FUNCTION_BLOCK StartProgramTask EXTENDS TcoUrRoboticsTask
VAR

	_stopType: TcoAbstractions.eTcoRoboticsStopType;
END_VAR



IF Execute() THEN
	_blink(inOnTime:=T#500MS,inOffTime:=T#500MS);

	IF _progress = 0 THEN
		IF NOT __ISVALIDREF(inoControl) THEN
			_varInfo :=__VARINFO(inoControl);
			Messenger.Programming(_sb.Clear().Append('<#Invalid reference: #>').Append(_varInfo.Symbol).ToString()).Pin();
		ELSIF NOT __ISVALIDREF(inoConfig) THEN                                                  
			_varInfo :=__VARINFO(inoConfig);                                                    
			Messenger.Programming(_sb.Clear().Append('<#Invalid reference: #>').Append(_varInfo.Symbol).ToString()).Pin();
		ELSIF NOT __ISVALIDREF(inoStatus) THEN                                                  
			_varInfo :=__VARINFO(inoStatus);                                                    
			Messenger.Programming(_sb.Clear().Append('<#Invalid reference: #>').Append(_varInfo.Symbol).ToString()).Pin();
			ELSE
			_progress := _progress + 1;
		END_IF

	END_IF
	IF _progress = 1 THEN
		inoControl.StartProgram:=_blink.outQ;
		_varInfo :=__VARINFO( inoStatus.State.CycleOn);                                                
		THIS^.Messenger.OnCondition(_infoTimer.Q AND NOT inoStatus.State.CycleOn).Warning(_sb.Clear().Append('<#Waiting for program running signal! #>').Append(_varInfo.Symbol).ToString());
		
		_varInfo :=__VARINFO( inoStatus.State.SystemInputBusy);                                                
		THIS^.Messenger.OnCondition(_infoTimer.Q AND  inoStatus.State.SystemInputBusy).Warning(_sb.Clear().Append('<#Waiting for system ready signal! #>').Append(_varInfo.Symbol).ToString());
		
		IF  inoStatus.State.CycleOn AND NOT inoStatus.State.SystemInputBusy THEN
				inoControl.StartProgram:=FALSE;
		END_IF
	END_IF;		
	
	

    DoneWhen(inoStatus.State.CycleOn );
    CallTimers(TRUE);
	
	THIS^.ThrowWhen(_errorTimer.Q OR inoStatus.State.Error);
END_IF

IF  THIS^.Error AND NOT _errorMessage.Pinned THEN
	THIS^.Restore();
END_IF

METHOD PUBLIC FB_init : BOOL
VAR_INPUT
    bInitRetains : BOOL; // if TRUE, the retain variables are initialized (warm start / cold start)
    bInCopyCode : BOOL; // if TRUE, the instance afterwards gets moved into the copy code (online change)
  	ParentObject : ITcoObject;	
END_VAR
END_METHOD

METHOD INTERNAL InvokeWithParams : ITcoTaskStatus
VAR_INPUT
	inStopType : eTcoRoboticsStopType;
END_VAR
_stopType := inStopType;
InvokeWithParams := THIS^.Invoke();
END_METHOD

(*~
	<docu>
		<summary>
			Executes when task is aborted.
		</summary>			
	</docu>	
~*)
METHOD PROTECTED OnAbort
IF  __ISVALIDREF(inoStatus) THEN   THIS^.inoStatus.ActionDescription := '<#Stop program was aborted, while not yet completed!#>';END_IF;
END_METHOD

(*~
	<docu>
		<summary>
			Executes when task reaches the ```Done``` state .
		</summary>			
	</docu>	
~*)
METHOD PROTECTED OnDone
IF  __ISVALIDREF(inoStatus) THEN  THIS^.inoStatus.ActionDescription := '<#Stop program was completed successfully.#>';END_IF; 
_progress:=0;
END_METHOD

(*~
	<docu>
		<summary>
			Executes when task reaches the ```Error``` state.
				</summary>			
	</docu>	
~*)
METHOD PROTECTED OnError
VAR
	description: STRING;
END_VAR
THIS^.inoStatus.ActionDescription := '<#Stopping program with error.#>'; 
IF  __ISVALIDREF(inoStatus) THEN   THIS^.inoStatus.ActionDescription := description; END_IF;
THIS^._errorMessage.Error(_sb.Clear().Append(description).Append(' To restore acknowledge this alarm.').ToString()).Pin();
END_METHOD

METHOD PROTECTED OnStart
IF  __ISVALIDREF(inoStatus) THEN  THIS^.inoStatus.ActionDescription := '<#Stopping program started.#>'; END_IF; 
CallTimers(FALSE);
END_METHOD

(*~
	<docu>
		<summary>
			Restores this instance to the Ready state. Can be called explicitly or from within one of the restore mechanisms.
			<para>
				See also <see cref="PlcDocu.TcoCore.TcoTask.AutoRestorable()"/>
			</para>
		</summary>			
	</docu>	
~*)
METHOD Restore : ITcoRestorable
SUPER^.Restore();
END_METHOD

END_FUNCTION_BLOCK

(* stored: Version 1.1.0.1, ProductVersion 3.1.4024.12
   POU StartProgramTask: Id {1230dcd3-a713-0d73-090f-6538260c7db5}, SpecialFunc None
   Method FB_init: Id {798593c7-bab7-0e23-3e40-693854c851c1}
   Method InvokeWithParams: Id {1018f4f3-e843-0eb9-0aa3-3c086c7a0fe8}
   Method OnAbort: Id {71688ea6-95a8-02ad-02e5-2806a6c2e741}
   Method OnDone: Id {39d8236d-db7c-0c4b-3971-cda791c81357}
   Method OnError: Id {0ef4edcc-4c48-0751-0d7f-ebf84c17c830}
   Method OnStart: Id {4eef4f24-3de6-0fb7-3a1f-b3e11e98fec7}
   Method Restore: Id {61895d9f-3ebe-0aeb-1d72-e60d224ff52e} *)
